TEXTLIST ProductType
  0 = '无' | Chinese: '无' | English: 'None' | Vietnamese: 'None'
  1 = '左线' | Chinese: '左线' | English: 'Left' | Vietnamese: 'Left'
  2 = '右线' | Chinese: '右线' | English: 'Right' | Vietnamese: 'Right'
   = ''
END_TEXTLIST

(* stored: Version 1.1.0.1, ProductVersion 3.1.4024.3
   TextList ProductType: Id {13607f26-3968-4ad0-ab92-a32ab6591329} *)
